FUNCTION Matrix_Product : Bool
VAR_IN_OUT CONSTANT
	A : Matrix;//left side matrix
	B : Matrix;//right side matrix
END_VAR
VAR_IN_OUT
	Res : Matrix;//must not be the same source as M_L or M_R
END_VAR
VAR
	Ri : UINT;
	Ci : UINT;
	I : UINT;
	Sum : LREAL;
END_VAR

IF NOT(Matrix_CanMult(A,B)) THEN
	Matrix_Product := FALSE;
	RETURN;
END_IF

IF A.Rows <> Res.Rows OR B.Cols <> Res.Cols THEN
	Matrix_Product := FALSE;
	RETURN;
END_IF

Matrix_Product := TRUE;

FOR Ri := 0 TO Res.Rows-1 DO
	FOR Ci := 0 TO Res.Cols-1 DO
		Sum := 0;
		FOR I := 0 TO A.Cols-1 DO
			Sum := Sum + A.GetRC(Ri,I) * B.GetRC(I,Ci);
		END_FOR
		Res.SetRC(Ri,Ci,Sum);
	END_FOR
END_FOR

END_FUNCTION

(* stored: Version 1.1.0.1, ProductVersion 3.1.4024.9
   POU Matrix_Product: Id {78d7729b-89b3-48bc-b06c-a73009771b2d}, SpecialFunc None *)
